{attribute 'qualified_only'}
TYPE E_ConfigurableCylinderCommand : (NONE := 0, TO_HOME := 1, TO_WORK := 2) DINT;
END_TYPE

(* stored: Version 1.1.0.1, ProductVersion 3.1.4024.12
   DUT E_ConfigurableCylinderCommand: Id {369077c9-e2e3-4ba8-b212-124e8c9169a4} *)
